TYPE sup_location:
    (s1_sup_location, s2_sup_location, s3_sup_location, s4_sup_location, s5_sup_location, s6_sup_location, s7_sup_location, s8_sup_location, s9_sup_location, s10_sup_location);
END_TYPE

(* stored: ProductVersion 3.1.0.18, Version 1.1.0.1 *)
